FUNCTION F_TO_MODBUS_REGISTER : WORD
VAR_INPUT
	S_INFO : S_MODBUS_REGISTER;
END_VAR
VAR
	ADDRESS_SPACE : POINTER TO WORD;
END_VAR

ADDRESS_SPACE := ADR(S_INFO.REGISTER_SPACE);
F_TO_MODBUS_REGISTER := ADDRESS_SPACE^ + S_INFO.REGISTER_OFFSET;

END_FUNCTION

(* stored: Version 1.1.0.1, ProductVersion 3.1.4020.3
   POU F_TO_MODBUS_REGISTER: Id {ef5d189e-35e3-460b-bff2-ac8839f9c8f1}, SpecialFunc None *)
